# EPICS autosave request: iocBoot/iocmmc100test/saveData.req
[prefix]
$(P)

[status]
$(P)saveData_status

[message]
$(P)saveData_message

[filename]
$(P)saveData_fileName

[counter]   # scan counter
$(P)saveData_scanNumber

[fileSystem] # scan file system
$(P)saveData_fileSystem

[subdir]    # scan file subdirectory
$(P)saveData_subDir

[fullPathName]
$(P)saveData_fullPathName

[realTime1D] # if nonzero, write 1D data as it comes in
$(P)saveData_realTime1D
